TYPE U_HW_OutputCommands :
UNION
	Commandregister: WORD;
	ByteOut0: BYTE;
	ByteOut1: BYTE;

END_UNION
END_TYPE

(* stored: Version 1.1.0.1, ProductVersion 3.1.4024.9
   DUT U_HW_OutputCommands: Id {753f8385-2b45-4832-be46-aca06882a313} *)
